(* CODESYS project oslomodell 3_2 BIRAVEEN.export

Project tree, tasks and I/O mapping:
  Device : CODESYS Control Win V3 x64, 3S - Smart Software Solutions GmbH, version 3.5.16.30
    application Application
      libraries: Standard, * (System); VisuDialogs, * (System)
      task MainTask (cyclic, interval 10 ms, priority 1) calls PLC_PRG
      task VISU_TASK (cyclic, interval 100 ms, priority 31) calls VisuElems.Visu_Prg
      function block Oslo_Modell_3 [ST]
      program PLC_PRG [CFC]
      visualisation Visualization
*)

// Device/Application/PLC_PRG
PROGRAM PLC_PRG
VAR
	Alarm_1: BOOL;
	Alarm_2: BOOL;
	Alarm_3: BOOL;
	Oslo_Modell: Oslo_Modell_3;
	V1: BOOL;
	V2: BOOL;
	V5: BOOL;
	Heater: BOOL;
	Resett: BOOL;
	Ref_V3: INT;
	Ref_V4: REAL;
	Tank_Level: REAL;
	Temp: REAL;
	Tempen: REAL;
	Outflowen: REAL;
	Inflowen: REAL;
	
	Tank_Level_High: BOOL;
	Tank_Level_Low: BOOL;

	Var2_ON: BOOL;
	Var3_ON: BOOL;

	V6_ON: BOOL;
	V6_ON1: BOOL;
END_VAR

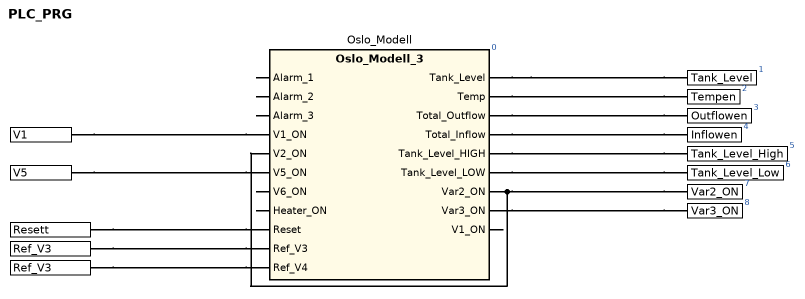
Oslo_Modell(
    V1_ON := V1,
    V2_ON := Oslo_Modell.Var2_ON,
    V5_ON := V5,
    Reset := Resett,
    Ref_V3 := Ref_V3,
    Ref_V4 := Ref_V3); // Oslo_Modell_3
Tank_Level := Oslo_Modell.Tank_Level;
Tempen := Oslo_Modell.Temp;
Outflowen := Oslo_Modell.Total_Outflow;
Inflowen := Oslo_Modell.Total_Inflow;
Tank_Level_High := Oslo_Modell.Tank_Level_HIGH;
Tank_Level_Low := Oslo_Modell.Tank_Level_LOW;
Var2_ON := Oslo_Modell.Var2_ON;
Var3_ON := Oslo_Modell.Var3_ON;

END_PROGRAM

// Device/Application/Oslo_Modell_3
FUNCTION_BLOCK Oslo_Modell_3

VAR_INPUT
	Alarm_1 : BOOL := FALSE;
	Alarm_2 : BOOL := FALSE;
	Alarm_3 : BOOL := FALSE;
	V1_ON : BOOL := FALSE;
	V2_ON : BOOL := FALSE;
	V5_ON : BOOL := FALSE;
	V6_ON : BOOL := FALSE;
	Heater_ON : BOOL := FALSE;
	Reset : BOOL := FALSE;
	Ref_V3 : REAL := 0;
	Ref_V4 : REAL := 0;	
END_VAR

VAR_OUTPUT
	Tank_Level : REAL := 30;
	Temp : REAL := 22;
	Total_Outflow : REAL := 0;
	Total_Inflow : REAL := 0;
	Tank_Level_HIGH : BOOL := FALSE;
	Tank_Level_LOW : BOOL := FALSE;
	Var2_ON: BOOL;
	Var3_ON: BOOL;
END_VAR
VAR
	Outflow : REAL := 0;
	Inflow : REAL := 0;
	
	Variabel_1: INT := 0;
END_VAR

IF NOT Reset THEN //Reset er FALSE
	IF V1_ON AND Ref_V3 > 49  THEN //Inflow ventilene er åpne
		IF Ref_V3 > 50 THEN //Den analoge ventilen er åpen
			Inflow := 0.05 + 0.0005*Ref_V3; //50% Inflow fra V5 + Inflow fra den analoge ventilen
		ELSE //Den analoge ventilen er stengt
			Inflow := 0.05; //50% Inflow fra V5
		END_IF
	ELSIF V1_ON AND Ref_V3 > 0 THEN //Hovedventilen er åpen og den analoge ventilen er åpen
		Inflow := 0.001*Ref_V3; //Inflow er proposjonal med verdien til ventilen
	ELSE
		Inflow := 0; 
	END_IF
	
	IF V2_ON AND Ref_V4 = Tank_Level THEN //Outflow ventilene er åpne
		IF Tank_Level <= 0 THEN
			Outflow := 0;
			Tank_Level := 0;
		ELSIF Ref_V4 > 50 THEN //Den analoge verdien er åpen
			Outflow := 0.05 + 0.0005*Ref_V4; //50% Inflow fra V6 + Outflow fra den analoge ventilen
		ELSE // Den analoge ventilen er stengt
			Outflow := 0.05; //50% Outflow fra V6
		END_IF
	ELSIF V2_ON AND Ref_V4 > 0 THEN //Hovedventilen er åpen og den analoge ventilen er åpen
		IF Tank_Level <= 0 THEN
			Outflow := 0;
			Tank_Level := 0;
		ELSE
		Outflow := 0.001*Ref_V4; //Outflow er proposjonal med verdien til ventilen
		END_IF
	ELSE
		Outflow := 0;
	END_IF
	
Tank_Level := Tank_Level + (Inflow - Outflow); //Tank nivået er en funksjon av Inflow - Outflow
Total_Outflow := Outflow*10;
Total_Inflow := Inflow*10;

	IF Tank_Level >= 90 THEN //Setter Tank_Level_HIGH om level er større enn 90
		Tank_Level_HIGH := TRUE;
	ELSE 
		Tank_Level_HIGH := FALSE;
	END_IF
	IF Tank_Level <= 10 THEN //Setter Tank_Level_LOW om level er mindre enn 10
		Tank_Level_LOW := TRUE; 
	ELSE 
		Tank_Level_LOW := FALSE;
	END_IF
	
	IF Heater_ON THEN //Varmeelementet er skrudd på
		Temp := Temp + (30000.0/(4187.0*Tank_Level)); //Temperaturen i tanken øker
	ELSE //Varmeelementet er av
		Temp := Temp - 0.04; //Temperaturen i tanken synker
		IF Temp <= 22 THEN //Sørger for at vannet ikke blir kaldere enn romtemperatur
			Temp := 22; //Sette temperaturen på vannet lik romtemperatur
		END_IF
	END_IF
		
ELSE //Reset er TRUE
// Resette variablene til initialverdier
	Ref_V3 := 50;
	Ref_V4 := 0;
	Temp := 22;
	Tank_Level := 30;
	V1_ON := FALSE;
	V2_ON := FALSE;
	V5_ON := FALSE;
	V6_ON := FALSE;
	Heater_ON := FALSE;
	Alarm_1 := FALSE;
	Alarm_2 := FALSE;
	Alarm_3 := FALSE;
	Tank_Level_HIGH := FALSE;
	Tank_level_LOW := FALSE;
	Var2_ON := FALSE;
	Var3_ON := FALSE;
	Variabel_1 := 0;

END_IF

IF Tank_Level >= 80 THEN
	Alarm_1 := TRUE;
END_IF

IF Tank_Level >= 80 THEN
	Var2_ON := TRUE;
END_IF
// OPPG 3_2
IF Tank_Level >= 80 AND Variabel_1 = 0 THEN
	Alarm_1 := TRUE;
	Variabel_1 := 2;
	V1_ON := FALSE;
	Heater_ON := TRUE;
END_IF

IF Temp >= 60  THEN
	Heater_ON := FALSE;
	Variabel_1 := 1;
END_IF

IF Temp < 50 AND Variabel_1 = 1 THEN
	Heater_ON := TRUE;
END_IF

END_FUNCTION_BLOCK

// Device/Application/Visualization
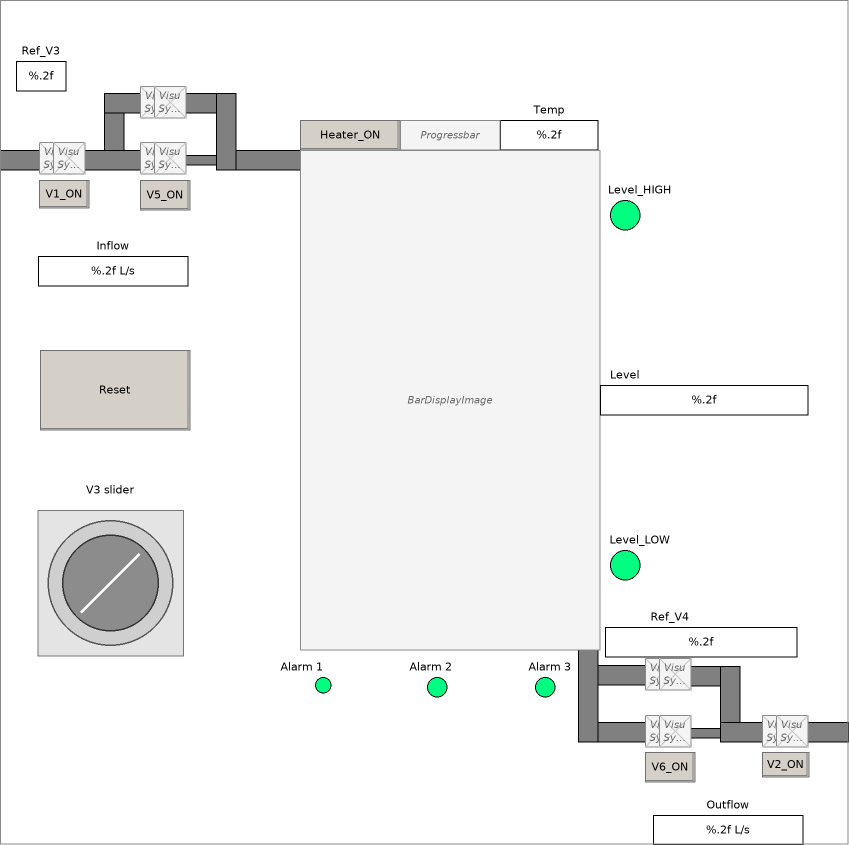
VISUALIZATION Visualization  // 849x845
    RoundedRectangle (104,101 20x60)
    Rectangle (500,120 98x30), "%.2f", text variable: PLC_PRG.Oslo_Modell.Temp
    Button (300,120 100x30), "Heater_ON"
        toggle PLC_PRG.Heater
    RoundedRectangle (682,666 45x20)
    RoundedRectangle (799,722 50x20)
    RoundedRectangle (580,722 77x20)
    RoundedRectangle (580,665 77x20)
    RoundedRectangle (578,642 20x100)
    RoundedRectangle (177,155 45x10)
    RoundedRectangle (227,150 82x20)
    RoundedRectangle (177,93 45x20)
    RoundedRectangle (216,93 20x77)
    RoundedRectangle (104,93 49x20)
    RoundedRectangle (77,150 75x20)
    BarDisplayImage (300,150 300x500), value: PLC_PRG.Oslo_Modell.Tank_Level, style: BarDisplayImage-Gray, scale format: %.1f, scale 0..100
    RoundedRectangle (0,150 50x20)
    Group (39,142 50x36)
        Image (0,0 32x32), image: VisuSymbols.Symbols.TriangleRight
        Image (14,0 32x32), image: VisuSymbols.Symbols.TriangleLeft
    Group (140,142 50x36)
        Image (0,0 32x32), image: VisuSymbols.Symbols.TriangleRight
        Image (14,0 32x32), image: VisuSymbols.Symbols.TriangleLeft
    Group (140,86 50x36)
        Image (0,0 32x32), image: VisuSymbols.Symbols.TriangleRight
        Image (14,0 32x32), image: VisuSymbols.Symbols.TriangleLeft
    Button (39,180 50x28), "V1_ON"
        toggle PLC_PRG.V1
    Button (140,180 50x30), "V5_ON"
        toggle PLC_PRG.V5
    Group (16,36 335x47)
        Rectangle (0,25 50x30), "%.2f", text variable: PLC_PRG.Oslo_Modell.Ref_V3
            OnMouseDown: write PLC_PRG.Oslo_Modell.Ref_V3 via InputWithLimits, min 0, max 100
        Label (0,0 50x30), "Ref_V3"
    Rectangle (600,385 208x30), "%.2f", text variable: PLC_PRG.Oslo_Modell.Tank_Level
    Ellipse (610,200 30x30), colour toggle: PLC_PRG.Oslo_Modell.Tank_Level_HIGH
    Ellipse (610,550 30x30), colour toggle: PLC_PRG.Oslo_Modell.Tank_Level_LOW
    Label (600,175 80x30), "Level_HIGH"
    Label (600,525 80x30), "Level_LOW"
    Label (600,360 50x30), "Level"
    Group (38,231 153x52), text variable: PLC_PRG.Oslo_Modell.Total_Inflow
        Rectangle (0,25 150x30), "%.2f L/s", text variable: PLC_PRG.Oslo_Modell.Total_Inflow
        Label (0,0 150x30), "Inflow"
    Button (40,350 150x80), "Reset"
        tap PLC_PRG.Resett
    RoundedRectangle (682,728 45x10)
    Group (645,658 50x36)
        Image (0,0 32x32), image: VisuSymbols.Symbols.TriangleRight
        Image (14,0 32x32), image: VisuSymbols.Symbols.TriangleLeft
    Group (645,715 50x36)
        Image (0,0 32x32), image: VisuSymbols.Symbols.TriangleRight
        Image (14,0 32x32), image: VisuSymbols.Symbols.TriangleLeft
    RoundedRectangle (720,666 20x72)
    RoundedRectangle (720,722 54x20)
    Group (762,715 50x36)
        Image (0,0 32x32), image: VisuSymbols.Symbols.TriangleRight
        Image (14,0 32x32), image: VisuSymbols.Symbols.TriangleLeft
    Button (645,752 50x30), "V6_ON"
        toggle PLC_PRG.V6_ON
    Button (762,752 47x25), "V2_ON"
    Rectangle (653,815 150x30), "%.2f L/s", text variable: PLC_PRG.Oslo_Modell.Total_Outflow
    Label (653,790 150x30), "Outflow"
    Rectangle (605,627 192x30), "%.2f", text variable: PLC_PRG.Oslo_Modell.Ref_V4
        OnMouseDown: write PLC_PRG.Oslo_Modell.Ref_V4 via InputWithLimits, min 0, max 100
    Label (645,602 50x30), "Ref_V4"
    Ellipse (315,677 16x16), colour toggle: PLC_PRG.Oslo_Modell.Alarm_1
        toggle PLC_PRG.Alarm_1
    Label (254,652 96x30), "Alarm 1"
    Ellipse (427,677 20x20), colour toggle: PLC_PRG.Oslo_Modell.Alarm_2
        toggle PLC_PRG.Alarm_2
    Label (388,652 86x30), "Alarm 2"
    Ellipse (535,677 20x20), colour toggle: PLC_PRG.Oslo_Modell.Alarm_3
        toggle PLC_PRG.Alarm_3
    Label (525,652 50x30), "Alarm 3"
    Progressbar (400,120 100x30), variable: PLC_PRG.Oslo_Modell.Temp
    Label (499,95 100x30), "Temp"
    Potentiometer360 (36,510 149x146), variable: PLC_PRG.Ref_V3, style: Potentiometer-Potentiometer360-Gray, scale format: %.1f, scale 0..100
        p2431819421: Outside
    Label (35,475 150x30), "V3 slider"
END_VISUALIZATION
